{attribute addProperty BoxType "KL9210"}
{attribute addProperty Id "Channel_1Channel_0970199100"}
{attribute addProperty CRC "2629167143"}
{attribute addProperty SizeInBites "0"}
{attribute addProperty SizeInBytes "0"}
TYPE KL9210_9CB5E827 :
STRUCT
	{attribute addProperty Name "Channel_1"}
	Channel_1 : Channel_09701991;
END_STRUCT
END_TYPE

(* stored: Version 1.2.0.0, ProductVersion 3.1.4024.9
   DUT KL9210_9CB5E827: Id {bf55a593-3c8a-4d6a-b127-e1fdcb798625} *)
